PROGRAM MAIN
VAR
END_VAR

Analogue_Processing();

END_PROGRAM

(* stored: Version 1.1.0.1, ProductVersion 3.1.4024.15
   POU MAIN: Id {4e25f483-92b0-4c03-b20f-252477a44d8d}, SpecialFunc None *)
